# EPICS substitutions: TRITON/TRITON-IOC-01App/Db/TRITON_pid.substitutions
file TRITON_pid.template {

pattern {PORT, P, CTRL}
{"\$(PORT)", "\$(P)", "P"}
{"\$(PORT)", "\$(P)", "I"}
{"\$(PORT)", "\$(P)", "D"}
}
